Fanuc KAREL source: kt00298.KL

-- PROVISIONAL review KL for V940-1; original PC SHA256 782eb3fea1d541c25fee0f0d233d733c49aedb5fb0c1a87d1a893d88b25f07b2
-- Incomplete behavior may be omitted. Consult companion uncertainty JSON. Do not deploy.
PROGRAM KT00298
%NOLOCKGROUP
VAR
  R1 : REAL
  R2 : REAL
  OUT : BOOLEAN
BEGIN
  -- V9_ZERO_TABLE_METADATA_HINT layout=0001; no indexed target words; source/name/runtime held
  -- UNRESOLVED_PC offsets 5-16; opcodes 2E,23
  -- UNRESOLVED_PC offsets 21-32; opcodes 2E,23
  -- UNRESOLVED_PC offsets 37-48; opcodes 2E,23
  -- UNRESOLVED_PC offsets 53-64; opcodes 2E,23
  -- UNRESOLVED_PC offsets 69-88; opcodes 21,21,6E,23
  -- UNRESOLVED_PC offsets 93-97; opcodes 7F
END KT00298
